FUNCTION_BLOCK E_CYCLE (* Peroidic event generator *)
  PACKAGE iec61499::events;
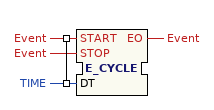
  EVENT_INPUT
    START WITH DT; (* Start the perodic generation of events *)
    STOP; (* Stop the generation of events *)
  END_EVENT
  EVENT_OUTPUT
    EO; (* Periodically triggered output event *)
  END_EVENT
  VAR_INPUT
    DT : TIME; (* cycle time *)
  END_VAR
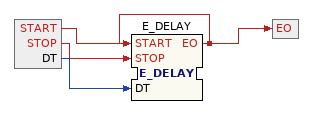
  FBS
    E_DELAY : iec61499::events::E_DELAY;
  END_FBS
  EVENT_CONNECTIONS
    START TO E_DELAY.START;
    STOP TO E_DELAY.STOP;
    E_DELAY.EO TO E_DELAY.START;
    E_DELAY.EO TO EO;
  END_CONNECTIONS
  DATA_CONNECTIONS
    DT TO E_DELAY.DT;
  END_CONNECTIONS
END_FUNCTION_BLOCK
